(* Logix 5000 project; controller DispersionPlc vendor 1 type 14 code 108 rev 34.11; software revision 34.01; part 7 of 22 *)
(* tags used below, declared in another part *)
   AllwaysOff : BOOL;
   BypassOns : BOOL;
   Dispertion_Intelock_Status : BOOL;
   DnEnable : BOOL;
   IntAlrTmr : TIMER[32];
   Inx_AlarmsResetting : BOOL;
   Inx_AlrResetIdx : DINT;
   Inx_NewAlarmScanIdx : DINT;
   inx_QuedAlarm : DINT;
   InxAckAlarms : BOOL[128];
   InxAlarmDisplayTmr : TIMER;
   NoNEwInxAlarmsDestedted : BOOL;
   ONS : BOOL[32];
   T4301_T4302_Xfer_In_Enable : BOOL;
   _JISdebug : DINT;
   _Placeholder : DINT;
   AFB : BOOL;
   AFI : BOOL;
   B4320_Transfer : BOOL;
   bypass_bit : BOOL;
   Cat_Man_ONS : BOOL;
   Cat_Pump_manual : BOOL;
   Dispersion_to_Main : DINT;
   Dispersion_to_SIL2 : DINT;
   Dispersion_to_SIL2_Analog : REAL[24];
   DispersionAlarms : BOOL[256];
   DPT_4320 : REAL;
   DPT_4320_High : REAL;
   DPT_4320_Raw : INT;
   Drum_Transfer : BOOL;
   Estop_Bulk : ALIAS FOR Local:1:I.Data[33].5;
   FQIC_4302_11_Pulse : BOOL;
   GasAlarmTmr : TIMER;
   GasAlarmTmrOff : TIMER;
   GasAlarmTmrOn : TIMER;
   Inx_AlarmScanIdx : DINT;
   Inx_Alr_To_Sound_Horn : BOOL[128];
   INX_ALRM_BUZ : ALIAS FOR Local:1:O.Data[1].9;
   InxAlarmResetBit : BOOL;
   InxAlarms : BOOL[128];
   LAH_4302_11 : BOOL;   // Truck Loading Level Alarm High Probe
   LevelAlarmBeaconsRelay : BOOL;
   LS_4320 : ALIAS FOR Local:1:I.Data[4].4;
   LS_T51_High : ALIAS FOR Local:1:I.Data[27].14;
   LVL_W2_High : ALIAS FOR Local:1:I.Data[1].22;
   LVL_W4_High : ALIAS FOR Local:1:I.Data[1].23;
   MCC1D4_20_TT5_Relay : BOOL;
   MCC1F3_TT1_Relay : BOOL;
   MCC1F4_8_TT9_Relay : BOOL;
   MCR_Bulk : ALIAS FOR Local:1:I.Data[33].4;
   MIXER_A_4320_AUX : ALIAS FOR Local:1:I.Data[1].5;
   MIXER_A_4320_RUN : ALIAS FOR Local:1:O.Data[0].5;
   MMI_7_8_Transfer_Pump_Start : BOOL;
   MMI_7_8_Transfer_Pump_Stop : BOOL;
   MMI_Cat_Man_Req : BOOL;
   MMI_Dispersion_Interlock_Bypass : BOOL;
   MMI_Dispersion_Interlock_Bypass_pb : BOOL;
   MMI_INX_Alarm_Reset_Pb : BOOL;
   MMI_INX_Solvent_Bypass_TOG : BOOL;
   MMI_Mon_Man_Req : BOOL;
   Mon_Man_ONS : BOOL;
   Mon_Pump_Manual : BOOL;
   NEW_TO : MESSAGE;
   OneShots : DINT;
   PS_AirMakeup : ALIAS FOR Local:1:I.Data[33].3;
   Pv_Inx_Alarm_Val : DINT;
   RG_T51 : REAL;
   RG_T51_Warn : REAL;
   RM_Pump_P51_Aux : ALIAS FOR Local:1:I.Data[33].2;
   RM_Pump_P51_Run : ALIAS FOR Local:1:O.Data[13].0;
   RM_Pump_P51_Run_PB : ALIAS FOR Local:1:I.Data[40].0;
   RM_Pump_P51_Run_PB_2 : ALIAS FOR Local:1:I.Data[40].2;
   RM_Tank_T51_Fill_Closed : ALIAS FOR Local:1:O.Data[12].10;
   RM_To_W2 : ALIAS FOR Local:1:I.Data[1].20;
   RM_To_W4 : ALIAS FOR Local:1:I.Data[1].21;
   SPARE_I306 : ALIAS FOR Local:3:I.Data.6;
   SPARE_I307 : ALIAS FOR Local:3:I.Data.7;
   SPARE_I308 : ALIAS FOR Local:3:I.Data.8;
   SPARE_I309 : ALIAS FOR Local:3:I.Data.9;
   SPARE_I310 : ALIAS FOR Local:3:I.Data.10;
   SPARE_I311 : ALIAS FOR Local:3:I.Data.11;
   SPARE_I312 : ALIAS FOR Local:3:I.Data.12;
   SPARE_I313 : ALIAS FOR Local:3:I.Data.13;
   SPARE_I314 : ALIAS FOR Local:3:I.Data.14;
   SPARE_I400 : ALIAS FOR Local:4:I.Data.0;
   SPARE_I401 : ALIAS FOR Local:4:I.Data.1;
   SPARE_I_1_1_18 : ALIAS FOR Local:1:I.Data[1].18;
   SPARE_I_1_1_19 : ALIAS FOR Local:1:I.Data[1].19;
   SPARE_O614 : ALIAS FOR Local:6:O.Data.14;
   SPARE_O615 : ALIAS FOR Local:6:O.Data.15;
   SPARE_O700 : ALIAS FOR Local:7:O.Data.0;
   SPARE_O701 : ALIAS FOR Local:7:O.Data.1;
   SPARE_O702 : ALIAS FOR Local:7:O.Data.2;
   SPARE_O703 : ALIAS FOR Local:7:O.Data.3;
   SPARE_O704 : ALIAS FOR Local:7:O.Data.4;
   SPARE_O705 : ALIAS FOR Local:7:O.Data.5;
   SPARE_O706 : ALIAS FOR Local:7:O.Data.6;
   SPARE_O707 : ALIAS FOR Local:7:O.Data.7;
   SPARE_O715 : ALIAS FOR Local:7:O.Data.15;
   SPARE_O_1_0_19 : ALIAS FOR Local:1:O.Data[0].19;
   SPARE_O_1_1_14 : ALIAS FOR Local:1:O.Data[1].14;
   SV_4303_03 : BOOL;
   SV_4303_04 : BOOL;
   SV_4304_02 : BOOL;
   SV_4304_03 : BOOL;
   T4301_Mixer : VFD;
   T4301_T4302_Xfer_In_Enable_Ctrl : BOOL;
   T52_Mixer : VFD;
   T53_Mixer : VFD;
   TE_4320 : INT;
   TE_4320_High : REAL;
   TOGGLE : BOOL;
   ToMesTmr : TIMER;
   TR_4320_Open : ALIAS FOR Local:1:I.Data[8].8;
   TRANS_PUMP_P_4320_AUX : ALIAS FOR Local:1:I.Data[1].6;
   TRANS_PUMP_P_4320_RUN : ALIAS FOR Local:1:O.Data[0].6;
   TruckLoadLevelAlarmResetPB : BOOL;
   TruckLoadLevelAlarmResetPBLight : BOOL;
   V4304_Pump : VFD;
   W4303_Pump : VFD;
   XV_4303_03 : BOOL;
   XV_4303_04 : BOOL;
   XV_4303_05 : BOOL;
   XV_4304_02 : BOOL;
   XV_4304_03 : BOOL;
   XV_4304_04 : BOOL;
   XV_4320_1 : ALIAS FOR Local:1:O.Data[1].1;
   XV_4320_2 : ALIAS FOR Local:1:O.Data[1].0;
   ZSC_4303_03 : BOOL;
   ZSC_4303_04 : BOOL;
   ZSC_4303_05 : BOOL;
   ZSC_4304_02 : BOOL;
   ZSC_4304_03 : BOOL;
   ZSC_4304_04 : BOOL;
   ZSC_4320_1 : ALIAS FOR Local:1:I.Data[4].3;
   ZSC_4320_2 : ALIAS FOR Local:1:I.Data[4].1;
   ZSO_4303_03 : BOOL;
   ZSO_4303_04 : BOOL;
   ZSO_4303_05 : BOOL;
   ZSO_4304_02 : BOOL;
   ZSO_4304_03 : BOOL;
   ZSO_4304_04 : BOOL;
   ZSO_4320_1 : ALIAS FOR Local:1:I.Data[4].2;
   ZSO_4320_2 : ALIAS FOR Local:1:I.Data[4].0;
(* MainProgram, continued *)

ROUTINE INX_Alarms   (* ladder *)
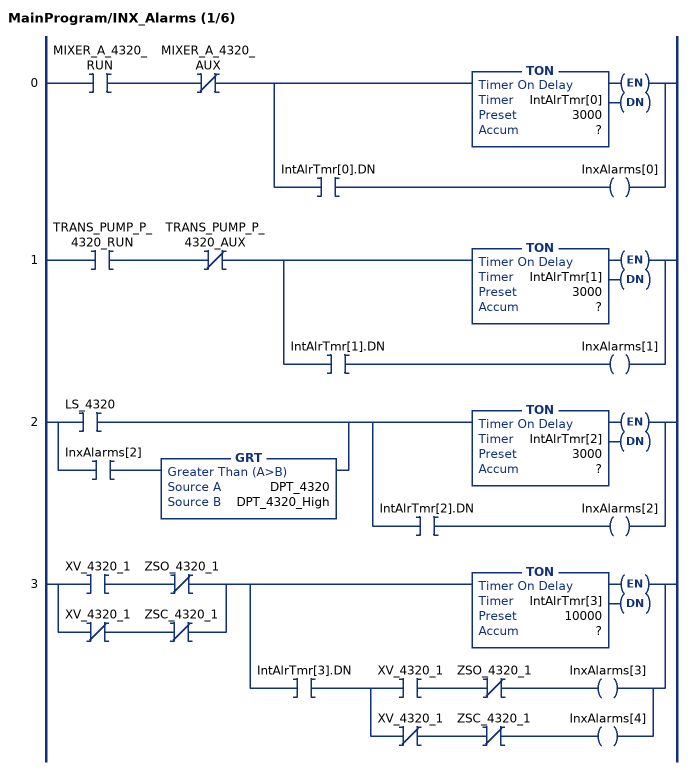
   0: XIC(MIXER_A_4320_RUN)XIO(MIXER_A_4320_AUX)[TON(IntAlrTmr[0],?,?) ,XIC(IntAlrTmr[0].DN) OTE(InxAlarms[0]) ];
   1: XIC(TRANS_PUMP_P_4320_RUN)XIO(TRANS_PUMP_P_4320_AUX)[TON(IntAlrTmr[1],?,?) ,XIC(IntAlrTmr[1].DN) OTE(InxAlarms[1]) ];
   2: [XIC(LS_4320) ,XIC(InxAlarms[2]) GRT(DPT_4320,DPT_4320_High) ][TON(IntAlrTmr[2],?,?) ,XIC(IntAlrTmr[2].DN) OTE(InxAlarms[2]) ];
   3: [XIC(XV_4320_1) XIO(ZSO_4320_1) ,XIO(XV_4320_1) XIO(ZSC_4320_1) ][TON(IntAlrTmr[3],?,?) ,XIC(IntAlrTmr[3].DN) [XIC(XV_4320_1) XIO(ZSO_4320_1) OTE(InxAlarms[3]) ,XIO(XV_4320_1) XIO(ZSC_4320_1) OTE(InxAlarms[4]) ] ];
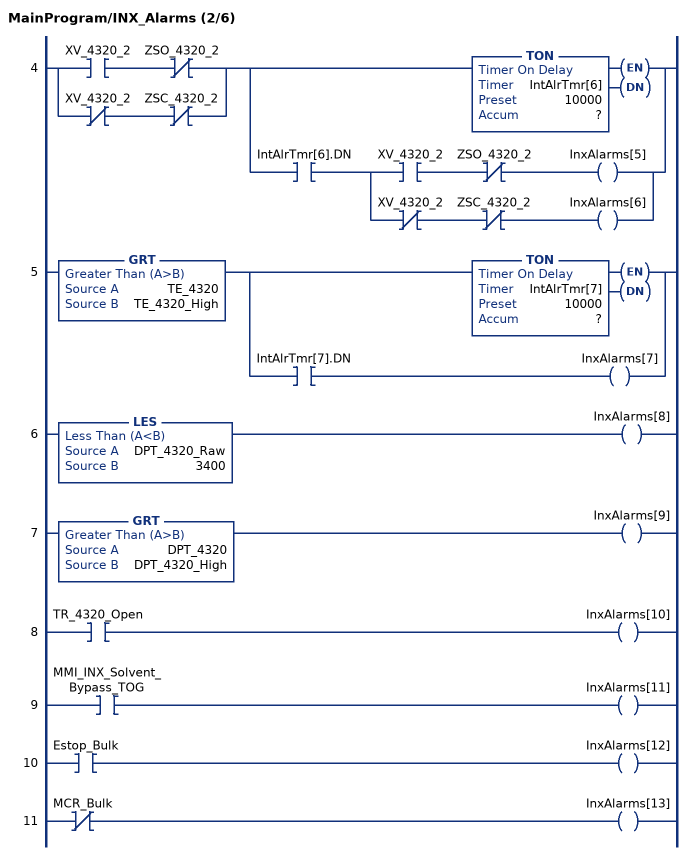
   4: [XIC(XV_4320_2) XIO(ZSO_4320_2) ,XIO(XV_4320_2) XIO(ZSC_4320_2) ][TON(IntAlrTmr[6],?,?) ,XIC(IntAlrTmr[6].DN) [XIC(XV_4320_2) XIO(ZSO_4320_2) OTE(InxAlarms[5]) ,XIO(XV_4320_2) XIO(ZSC_4320_2) OTE(InxAlarms[6]) ] ];
   5: GRT(TE_4320,TE_4320_High)[TON(IntAlrTmr[7],?,?) ,XIC(IntAlrTmr[7].DN) OTE(InxAlarms[7]) ];
   6: LES(DPT_4320_Raw,3400)OTE(InxAlarms[8]);
   7: GRT(DPT_4320,DPT_4320_High)OTE(InxAlarms[9]);
   8: XIC(TR_4320_Open)OTE(InxAlarms[10]);
   9: XIC(MMI_INX_Solvent_Bypass_TOG)OTE(InxAlarms[11]);
   10: XIC(Estop_Bulk)OTE(InxAlarms[12]);
   11: XIO(MCR_Bulk)OTE(InxAlarms[13]);
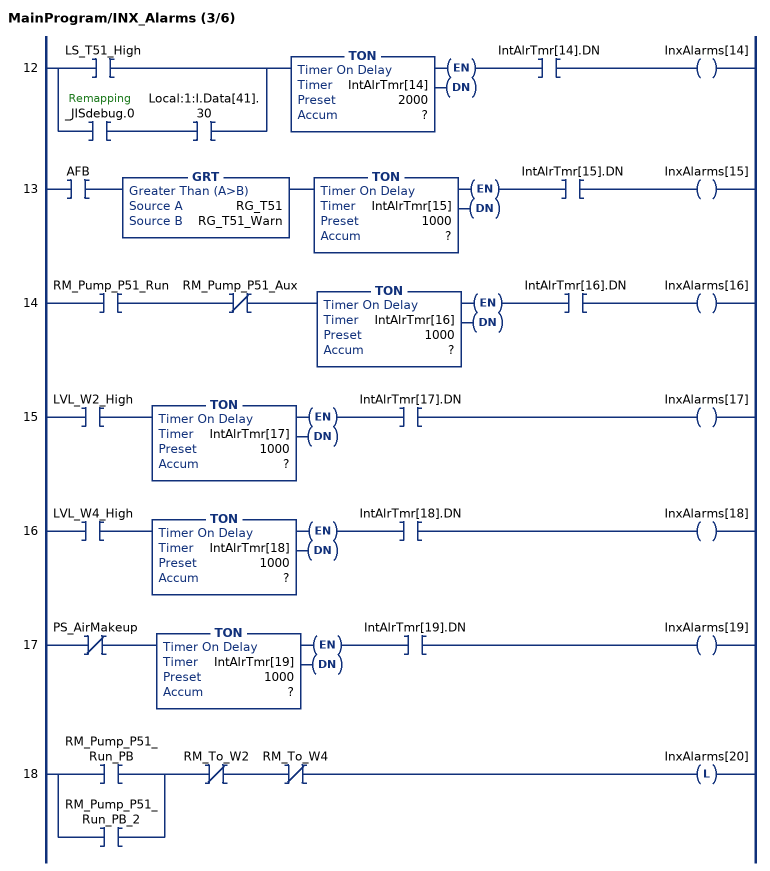
   12: [XIC(LS_T51_High) ,XIC(_JISdebug.0) XIC(Local:1:I.Data[41].30) ]TON(IntAlrTmr[14],?,?)XIC(IntAlrTmr[14].DN)OTE(InxAlarms[14]);
   13: XIC(AFB)GRT(RG_T51,RG_T51_Warn)TON(IntAlrTmr[15],?,?)XIC(IntAlrTmr[15].DN)OTE(InxAlarms[15]);
   14: XIC(RM_Pump_P51_Run)XIO(RM_Pump_P51_Aux)TON(IntAlrTmr[16],?,?)XIC(IntAlrTmr[16].DN)OTE(InxAlarms[16]);
   15: XIC(LVL_W2_High)TON(IntAlrTmr[17],?,?)XIC(IntAlrTmr[17].DN)OTE(InxAlarms[17]);
   16: XIC(LVL_W4_High)TON(IntAlrTmr[18],?,?)XIC(IntAlrTmr[18].DN)OTE(InxAlarms[18]);
   17: XIO(PS_AirMakeup)TON(IntAlrTmr[19],?,?)XIC(IntAlrTmr[19].DN)OTE(InxAlarms[19]);
   18: [XIC(RM_Pump_P51_Run_PB) ,XIC(RM_Pump_P51_Run_PB_2) ]XIO(RM_To_W2)XIO(RM_To_W4)OTL(InxAlarms[20]);
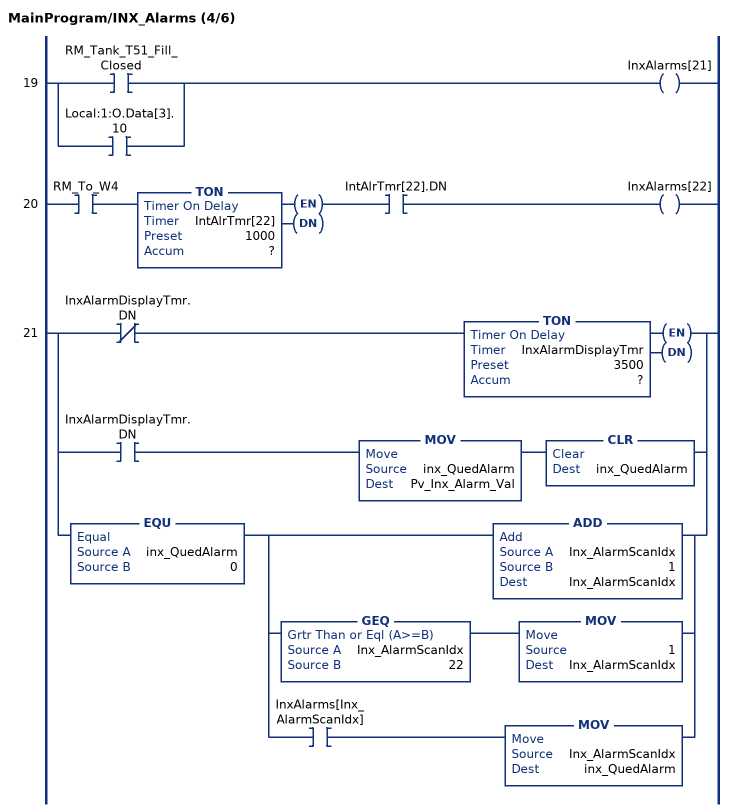
   19: [XIC(RM_Tank_T51_Fill_Closed) ,XIC(Local:1:O.Data[3].10) ]OTE(InxAlarms[21]);
   20: XIC(RM_To_W4)TON(IntAlrTmr[22],?,?)XIC(IntAlrTmr[22].DN)OTE(InxAlarms[22]);
   21: [XIO(InxAlarmDisplayTmr.DN) TON(InxAlarmDisplayTmr,?,?) ,XIC(InxAlarmDisplayTmr.DN) MOV(inx_QuedAlarm,Pv_Inx_Alarm_Val) CLR(inx_QuedAlarm) ,EQU(inx_QuedAlarm,0) [ADD(Inx_AlarmScanIdx,1,Inx_AlarmScanIdx) ,GEQ(Inx_AlarmScanIdx,22) MOV(1,Inx_AlarmScanIdx) ,XIC(InxAlarms[Inx_AlarmScanIdx]) MOV(Inx_AlarmScanIdx,inx_QuedAlarm) ] ];
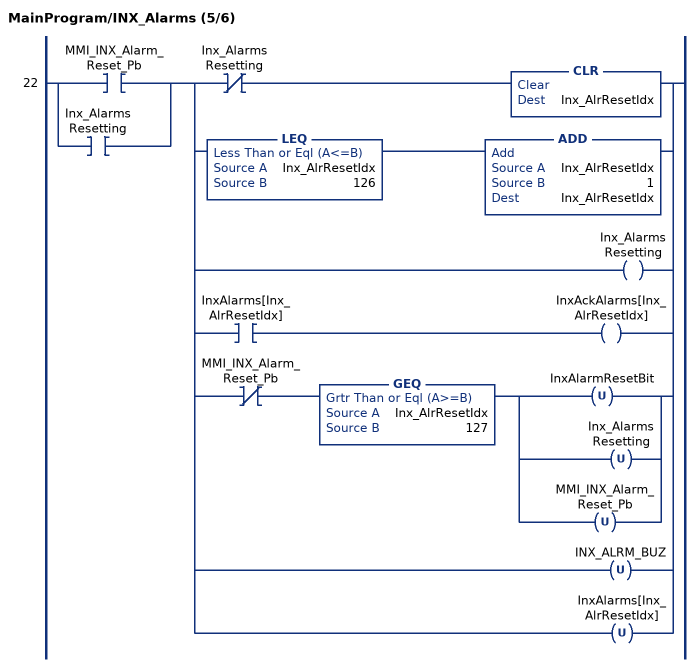
   22: [XIC(MMI_INX_Alarm_Reset_Pb) ,XIC(Inx_AlarmsResetting) ][XIO(Inx_AlarmsResetting) CLR(Inx_AlrResetIdx) ,LEQ(Inx_AlrResetIdx,126) ADD(Inx_AlrResetIdx,1,Inx_AlrResetIdx) ,OTE(Inx_AlarmsResetting) ,XIC(InxAlarms[Inx_AlrResetIdx]) OTE(InxAckAlarms[Inx_AlrResetIdx]) ,XIO(MMI_INX_Alarm_Reset_Pb) GEQ(Inx_AlrResetIdx,127) [OTU(InxAlarmResetBit) ,OTU(Inx_AlarmsResetting) ,OTU(MMI_INX_Alarm_Reset_Pb) ] ,OTU(INX_ALRM_BUZ) ,OTU(InxAlarms[Inx_AlrResetIdx]) ];
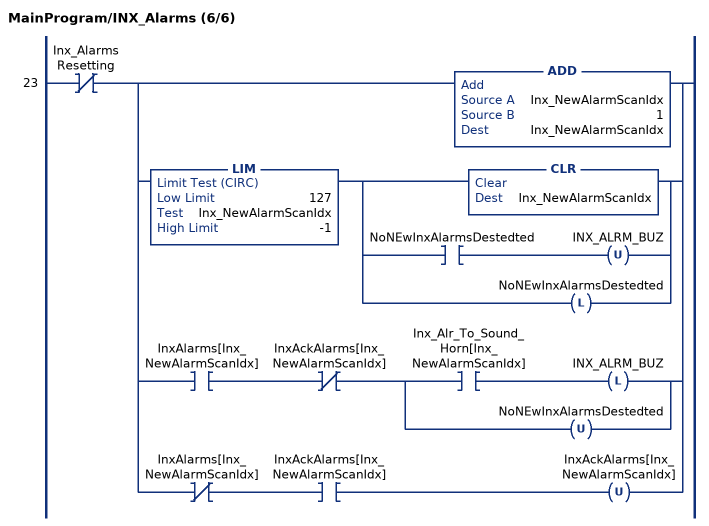
   23: XIO(Inx_AlarmsResetting)[ADD(Inx_NewAlarmScanIdx,1,Inx_NewAlarmScanIdx) ,LIM(127,Inx_NewAlarmScanIdx,-1) [CLR(Inx_NewAlarmScanIdx) ,XIC(NoNEwInxAlarmsDestedted) OTU(INX_ALRM_BUZ) ,OTL(NoNEwInxAlarmsDestedted) ] ,XIC(InxAlarms[Inx_NewAlarmScanIdx]) XIO(InxAckAlarms[Inx_NewAlarmScanIdx]) [XIC(Inx_Alr_To_Sound_Horn[Inx_NewAlarmScanIdx]) OTL(INX_ALRM_BUZ) ,OTU(NoNEwInxAlarmsDestedted) ] ,XIO(InxAlarms[Inx_NewAlarmScanIdx]) XIC(InxAckAlarms[Inx_NewAlarmScanIdx]) OTU(InxAckAlarms[Inx_NewAlarmScanIdx]) ];
END_ROUTINE

ROUTINE MainRoutine   (* ladder *)
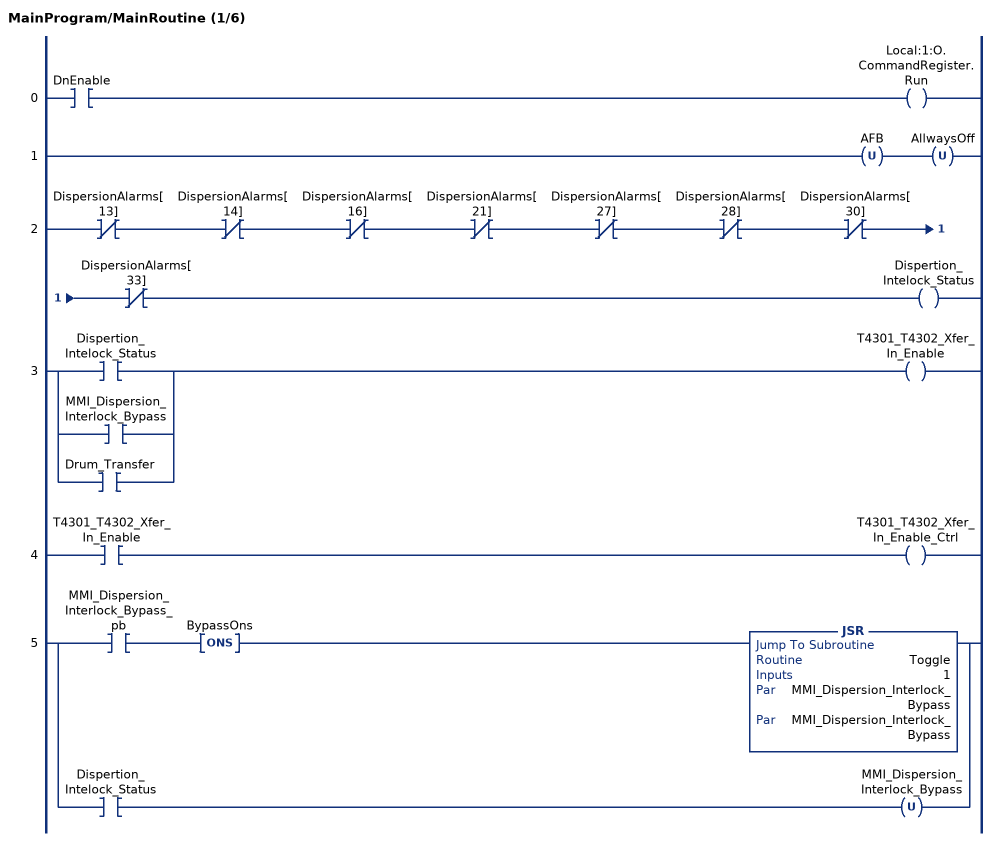
   0: XIC(DnEnable)OTE(Local:1:O.CommandRegister.Run);
   1: OTU(AFB)OTU(AllwaysOff);
   2: XIO(DispersionAlarms[13])XIO(DispersionAlarms[14])XIO(DispersionAlarms[16])XIO(DispersionAlarms[21])XIO(DispersionAlarms[27])XIO(DispersionAlarms[28])XIO(DispersionAlarms[30])XIO(DispersionAlarms[33])OTE(Dispertion_Intelock_Status);
   3: [XIC(Dispertion_Intelock_Status) ,XIC(MMI_Dispersion_Interlock_Bypass) ,XIC(Drum_Transfer) ]OTE(T4301_T4302_Xfer_In_Enable);
   4: XIC(T4301_T4302_Xfer_In_Enable)OTE(T4301_T4302_Xfer_In_Enable_Ctrl);
   5: [XIC(MMI_Dispersion_Interlock_Bypass_pb) ONS(BypassOns) JSR(Toggle,1,MMI_Dispersion_Interlock_Bypass,MMI_Dispersion_Interlock_Bypass) ,XIC(Dispertion_Intelock_Status) OTU(MMI_Dispersion_Interlock_Bypass) ];
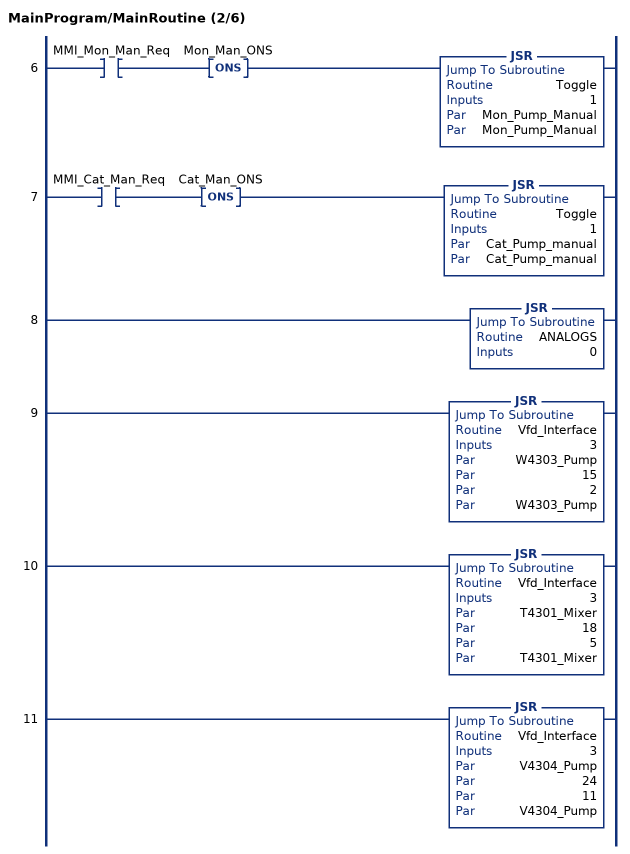
   6: XIC(MMI_Mon_Man_Req)ONS(Mon_Man_ONS)JSR(Toggle,1,Mon_Pump_Manual,Mon_Pump_Manual);
   7: XIC(MMI_Cat_Man_Req)ONS(Cat_Man_ONS)JSR(Toggle,1,Cat_Pump_manual,Cat_Pump_manual);
   8: JSR(ANALOGS,0);
   9: JSR(Vfd_Interface,3,W4303_Pump,15,2,W4303_Pump);
   10: JSR(Vfd_Interface,3,T4301_Mixer,18,5,T4301_Mixer);
   11: JSR(Vfd_Interface,3,V4304_Pump,24,11,V4304_Pump);
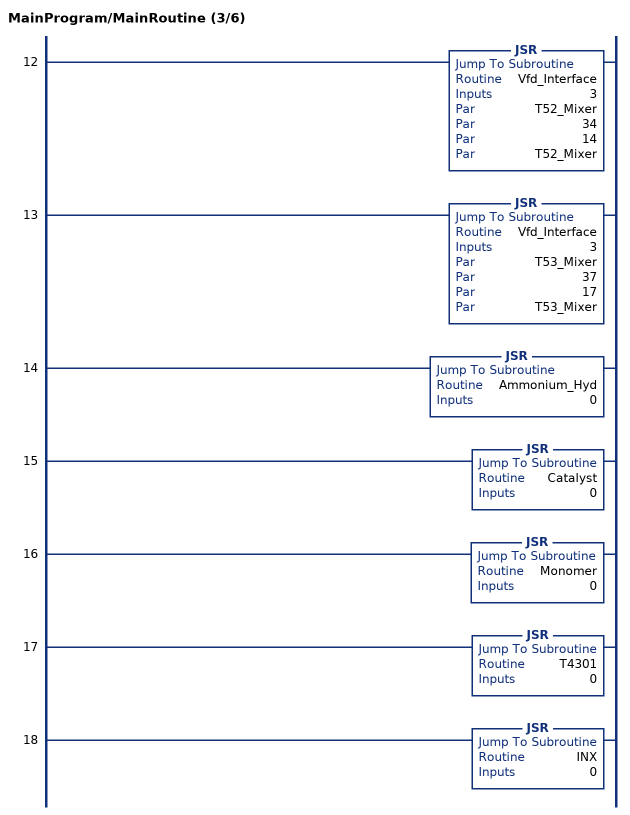
   12: JSR(Vfd_Interface,3,T52_Mixer,34,14,T52_Mixer);
   13: JSR(Vfd_Interface,3,T53_Mixer,37,17,T53_Mixer);
   14: JSR(Ammonium_Hyd,0);
   15: JSR(Catalyst,0);
   16: JSR(Monomer,0);
   17: JSR(T4301,0);
   18: JSR(INX,0);
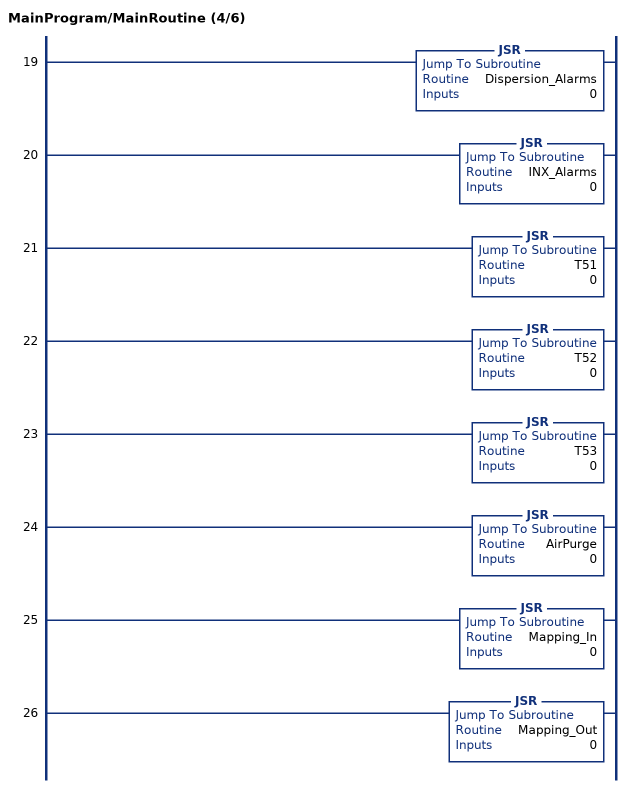
   19: JSR(Dispersion_Alarms,0);
   20: JSR(INX_Alarms,0);
   21: JSR(T51,0);
   22: JSR(T52,0);
   23: JSR(T53,0);
   24: JSR(AirPurge,0);
   25: JSR(Mapping_In,0);
   26: JSR(Mapping_Out,0);
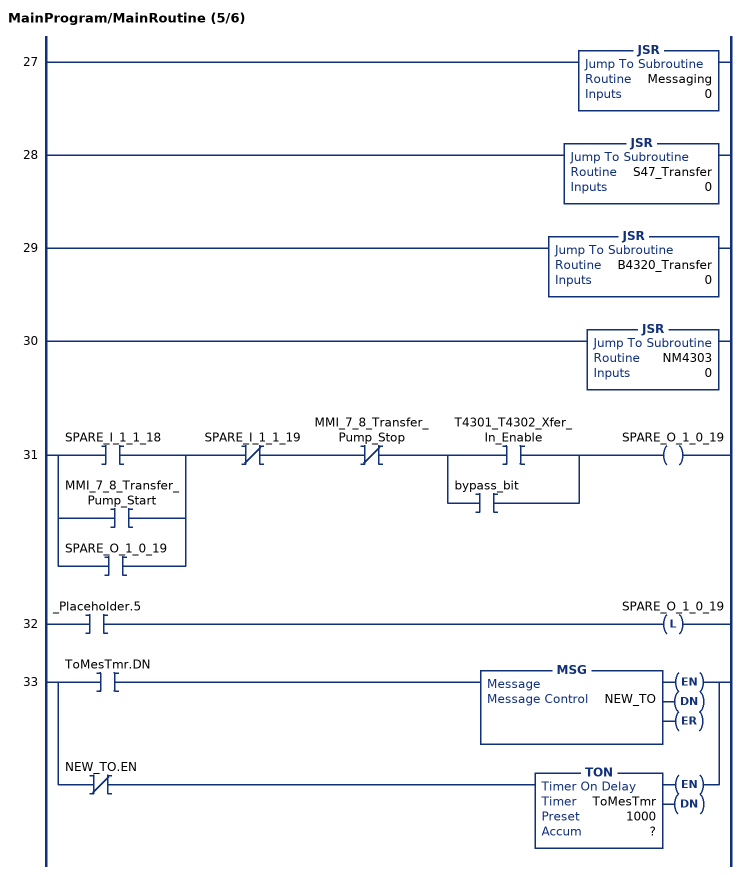
   27: JSR(Messaging,0);
   28: JSR(S47_Transfer,0);
   29: JSR(B4320_Transfer,0);
   30: JSR(NM4303,0);
   31: [[XIC(SPARE_I_1_1_18) ,XIC(MMI_7_8_Transfer_Pump_Start) ] ,XIC(SPARE_O_1_0_19) ]XIO(SPARE_I_1_1_19)XIO(MMI_7_8_Transfer_Pump_Stop)[XIC(T4301_T4302_Xfer_In_Enable) ,XIC(bypass_bit) ]OTE(SPARE_O_1_0_19);
   32: XIC(_Placeholder.5)OTL(SPARE_O_1_0_19);
   33: [XIC(ToMesTmr.DN) MSG(NEW_TO) ,XIO(NEW_TO.EN) TON(ToMesTmr,?,?) ];
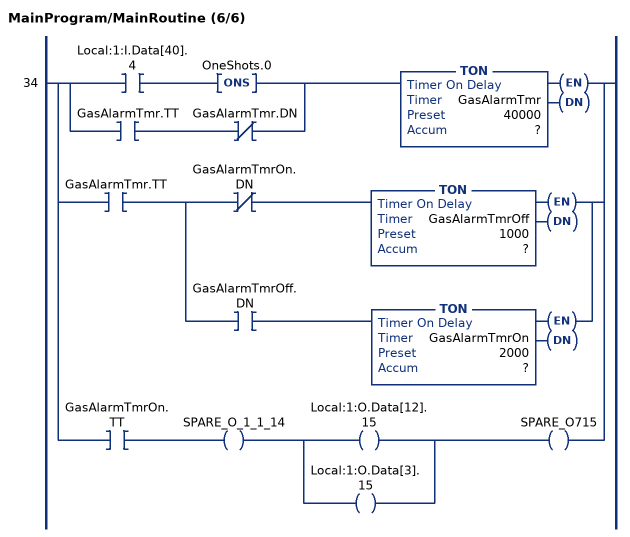
   34: [[XIC(Local:1:I.Data[40].4) ONS(OneShots.0) ,XIC(GasAlarmTmr.TT) XIO(GasAlarmTmr.DN) ] TON(GasAlarmTmr,?,?) ,XIC(GasAlarmTmr.TT) [XIO(GasAlarmTmrOn.DN) TON(GasAlarmTmrOff,?,?) ,XIC(GasAlarmTmrOff.DN) TON(GasAlarmTmrOn,?,?) ] ,XIC(GasAlarmTmrOn.TT) OTE(SPARE_O_1_1_14) [OTE(Local:1:O.Data[12].15) ,OTE(Local:1:O.Data[3].15) ] OTE(SPARE_O715) ];
END_ROUTINE

ROUTINE Mapping_In   (* ladder *)
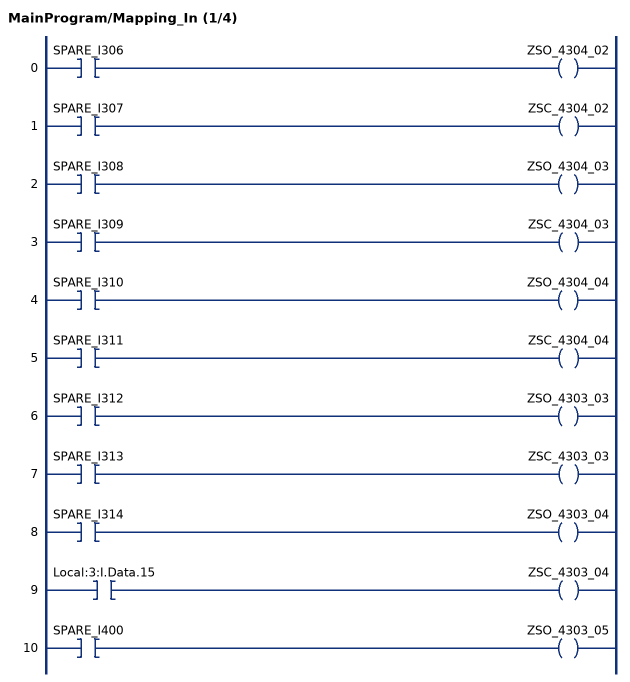
   0: XIC(SPARE_I306)OTE(ZSO_4304_02);
   1: XIC(SPARE_I307)OTE(ZSC_4304_02);
   2: XIC(SPARE_I308)OTE(ZSO_4304_03);
   3: XIC(SPARE_I309)OTE(ZSC_4304_03);
   4: XIC(SPARE_I310)OTE(ZSO_4304_04);
   5: XIC(SPARE_I311)OTE(ZSC_4304_04);
   6: XIC(SPARE_I312)OTE(ZSO_4303_03);
   7: XIC(SPARE_I313)OTE(ZSC_4303_03);
   8: XIC(SPARE_I314)OTE(ZSO_4303_04);
   9: XIC(Local:3:I.Data.15)OTE(ZSC_4303_04);
   10: XIC(SPARE_I400)OTE(ZSO_4303_05);
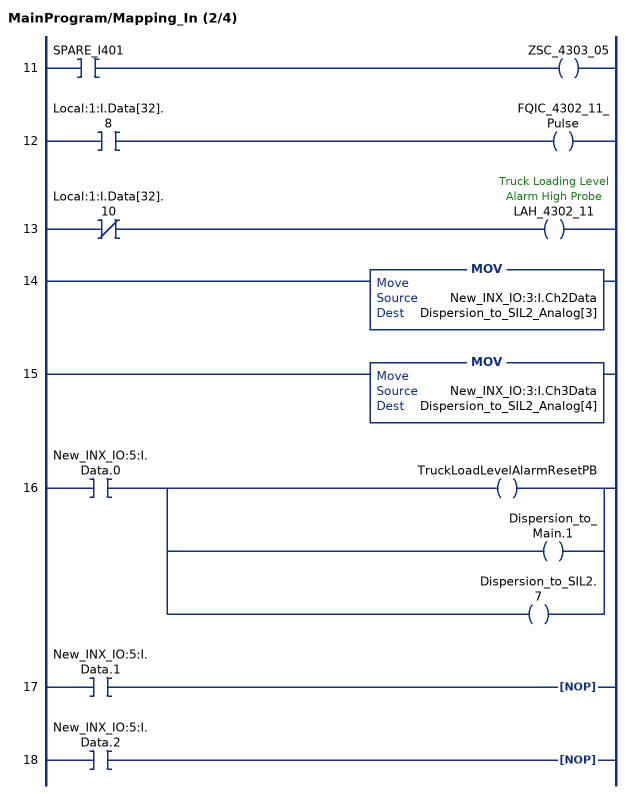
   11: XIC(SPARE_I401)OTE(ZSC_4303_05);
   12: XIC(Local:1:I.Data[32].8)OTE(FQIC_4302_11_Pulse);
   13: XIO(Local:1:I.Data[32].10)OTE(LAH_4302_11);
   14: MOV(New_INX_IO:3:I.Ch2Data,Dispersion_to_SIL2_Analog[3]);
   15: MOV(New_INX_IO:3:I.Ch3Data,Dispersion_to_SIL2_Analog[4]);
   16: XIC(New_INX_IO:5:I.Data.0)[OTE(TruckLoadLevelAlarmResetPB) ,OTE(Dispersion_to_Main.1) ,OTE(Dispersion_to_SIL2.7) ];
   17: XIC(New_INX_IO:5:I.Data.1)NOP();
   18: XIC(New_INX_IO:5:I.Data.2)NOP();
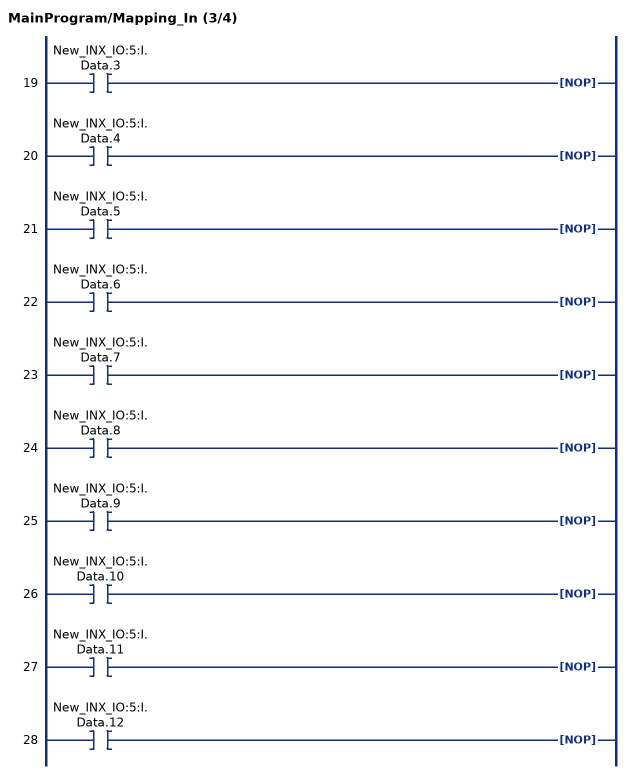
   19: XIC(New_INX_IO:5:I.Data.3)NOP();
   20: XIC(New_INX_IO:5:I.Data.4)NOP();
   21: XIC(New_INX_IO:5:I.Data.5)NOP();
   22: XIC(New_INX_IO:5:I.Data.6)NOP();
   23: XIC(New_INX_IO:5:I.Data.7)NOP();
   24: XIC(New_INX_IO:5:I.Data.8)NOP();
   25: XIC(New_INX_IO:5:I.Data.9)NOP();
   26: XIC(New_INX_IO:5:I.Data.10)NOP();
   27: XIC(New_INX_IO:5:I.Data.11)NOP();
   28: XIC(New_INX_IO:5:I.Data.12)NOP();
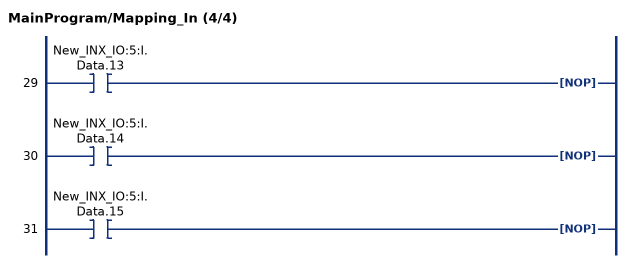
   29: XIC(New_INX_IO:5:I.Data.13)NOP();
   30: XIC(New_INX_IO:5:I.Data.14)NOP();
   31: XIC(New_INX_IO:5:I.Data.15)NOP();
END_ROUTINE

ROUTINE Mapping_Out   (* ladder *)
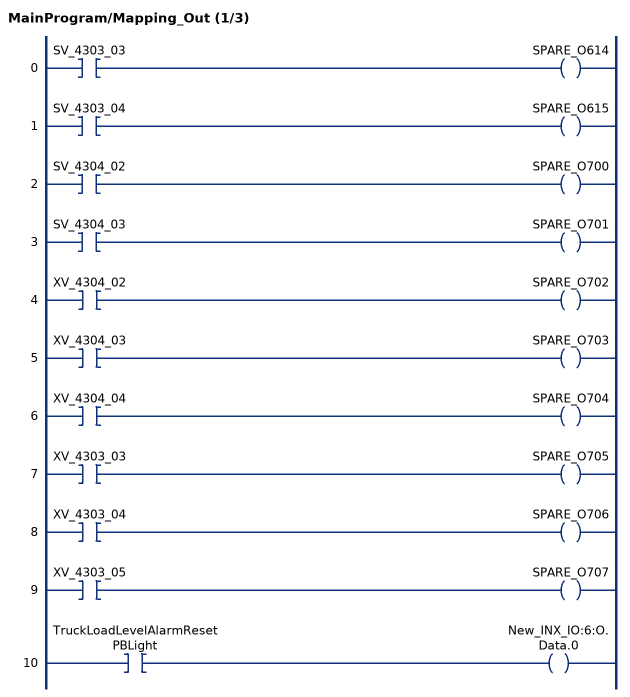
   0: XIC(SV_4303_03)OTE(SPARE_O614);
   1: XIC(SV_4303_04)OTE(SPARE_O615);
   2: XIC(SV_4304_02)OTE(SPARE_O700);
   3: XIC(SV_4304_03)OTE(SPARE_O701);
   4: XIC(XV_4304_02)OTE(SPARE_O702);
   5: XIC(XV_4304_03)OTE(SPARE_O703);
   6: XIC(XV_4304_04)OTE(SPARE_O704);
   7: XIC(XV_4303_03)OTE(SPARE_O705);
   8: XIC(XV_4303_04)OTE(SPARE_O706);
   9: XIC(XV_4303_05)OTE(SPARE_O707);
   10: XIC(TruckLoadLevelAlarmResetPBLight)OTE(New_INX_IO:6:O.Data.0);
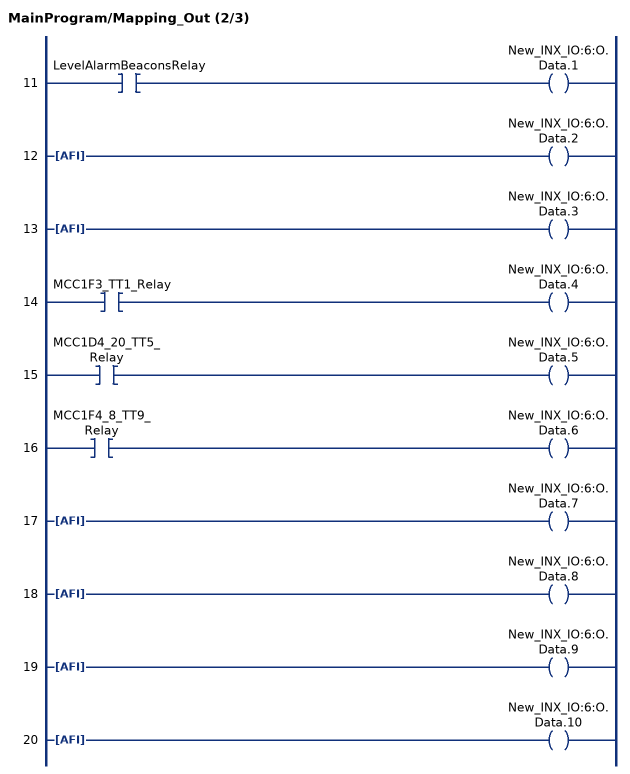
   11: XIC(LevelAlarmBeaconsRelay)OTE(New_INX_IO:6:O.Data.1);
   12: AFI()OTE(New_INX_IO:6:O.Data.2);
   13: AFI()OTE(New_INX_IO:6:O.Data.3);
   14: XIC(MCC1F3_TT1_Relay)OTE(New_INX_IO:6:O.Data.4);
   15: XIC(MCC1D4_20_TT5_Relay)OTE(New_INX_IO:6:O.Data.5);
   16: XIC(MCC1F4_8_TT9_Relay)OTE(New_INX_IO:6:O.Data.6);
   17: AFI()OTE(New_INX_IO:6:O.Data.7);
   18: AFI()OTE(New_INX_IO:6:O.Data.8);
   19: AFI()OTE(New_INX_IO:6:O.Data.9);
   20: AFI()OTE(New_INX_IO:6:O.Data.10);
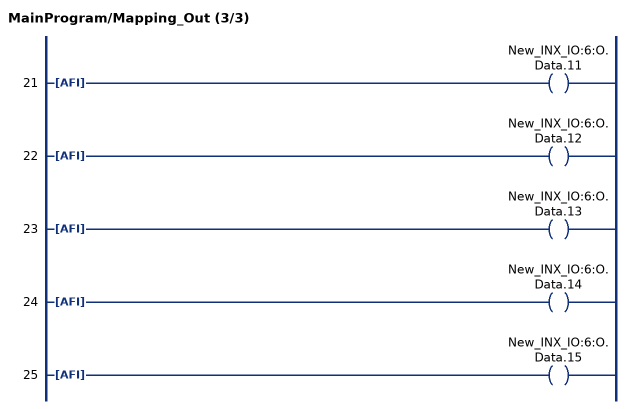
   21: AFI()OTE(New_INX_IO:6:O.Data.11);
   22: AFI()OTE(New_INX_IO:6:O.Data.12);
   23: AFI()OTE(New_INX_IO:6:O.Data.13);
   24: AFI()OTE(New_INX_IO:6:O.Data.14);
   25: AFI()OTE(New_INX_IO:6:O.Data.15);
END_ROUTINE
